FUNCTION_BLOCK ABSTRACT FB_Test IMPLEMENTS ITest
VAR
END_VAR

METHOD PROTECTED AssertEquals : ST_TestResults
VAR_INPUT
	expected		: ANY;
	result			: ANY;
	failmsg			: STRING(255);
END_VAR
VAR
	sExp, sRes		: STRING;
	results			: ST_TestResults;
END_VAR
IF (expected.diSize <> result.diSize) THEN
	results.Message := 'Test error: expected value type mismatch';
	results.Result := FALSE;
	AssertEquals := results;
	RETURN;
END_IF

IF (Expected.pValue^ <> Result.pValue^) THEN
	sExp := CONCAT(' Expected: ', TO_STRING(expected.pValue^));
	sRes := CONCAT(' Result: ', TO_STRING(result.pValue^));
	results.Message := CONCAT(CONCAT(failmsg, sExp), sRes);
	results.Result := FALSE;
	AssertEquals := results;
ELSE
	results.Result := TRUE;
	AssertEquals := results;
END_IF
END_METHOD

{attribute 'TcRpcEnable'}
METHOD Execute : ST_TestResults;
VAR
END_VAR
END_METHOD

END_FUNCTION_BLOCK

(* stored: Version 1.1.0.1, ProductVersion 3.1.4024.12
   POU FB_Test: Id {8831bd5e-bd34-44b6-83a6-6d659c4588f7}, SpecialFunc None
   Method AssertEquals: Id {b7f9f968-56cb-477a-b18f-fd7d7ae6de0b}
   Method Execute: Id {935cc836-92fd-4164-acc4-799697454b33} *)
